(* CODESYS project FU_sConcat9BIBO.xml

Project tree, tasks and I/O mapping:
  function FU_sConcat9BIBO [ST]
*)

// FU_sConcat9BIBO
//This functions combines nine strings
//This is the big output version, it has no limits to input or output size
//The wOutSize must be correct otherwise the function can write to unwanted addresses
// |**Version**|**Author**| **Date** |**Changes**
// | 1         | NSN      | 05-02-19 | Creation
// | 2         | NSN      | 14-10-21 | Changed to pointer based
FUNCTION FU_sConcat9BIBO : BOOL
VAR_INPUT
	sOut		:POINTER TO EASCII;			//Output String
	s1			:POINTER TO EASCII;			//Input String1
	s2			:POINTER TO EASCII;			//Input String2
	s3			:POINTER TO EASCII;			//Input String3
	s4			:POINTER TO EASCII;			//Input String4
	s5			:POINTER TO EASCII;			//Input String5
	s6			:POINTER TO EASCII;			//Input String6
	s7			:POINTER TO EASCII;			//Input String7
	s8			:POINTER TO EASCII;			//Input String8
	s9			:POINTER TO EASCII;			//Input String9
END_VAR
VAR_INPUT
	wOutSize	:WORD;				//Output String Size
END_VAR

WHILE wOutSize > 0 DO
	wOutSize		:=		wOutSize - 1;
	IF s1^ <> 0 THEN
		sOut^		:=		s1^;
		s1			:=		s1 + 1;
	ELSIF s2^ <> 0 THEN
		sOut^		:=		s2^;
		s2			:=		s2 + 1;
	ELSIF s3^ <> 0 THEN
		sOut^		:=		s3^;
		s3			:=		s3 + 1;
	ELSIF s4^ <> 0 THEN
		sOut^		:=		s4^;
		s4			:=		s4 + 1;
	ELSIF s5^ <> 0 THEN
		sOut^		:=		s5^;
		s5			:=		s5 + 1;
	ELSIF s6^ <> 0 THEN
		sOut^		:=		s6^;
		s6			:=		s6 + 1;
	ELSIF s7^ <> 0 THEN
		sOut^		:=		s7^;
		s7			:=		s7 + 1;
	ELSIF s8^ <> 0 THEN
		sOut^		:=		s8^;
		s8			:=		s8 + 1;
	ELSIF s9^ <> 0 THEN
		sOut^		:=		s9^;
		s9			:=		s9 + 1;
	ELSE
		EXIT;
	END_IF
	sOut			:=		sOut + 1;
END_WHILE
sOut^				:=		EASCII.Null;

END_FUNCTION
